RoboDK station: finished_products_shelf.rdk

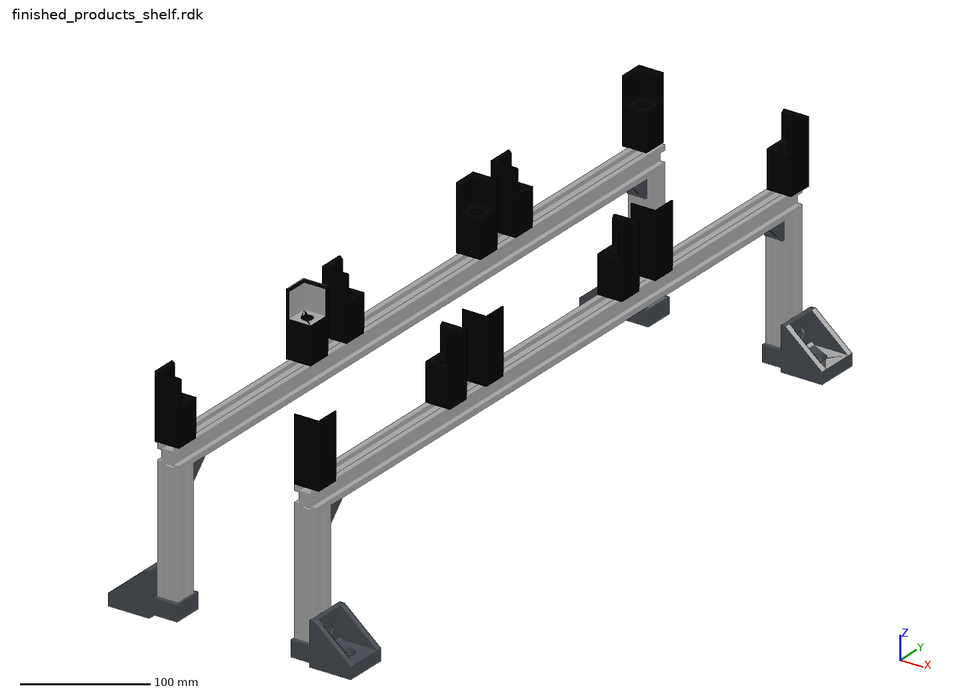
[picture v0: the station drawn from its stored meshes, robots at their saved joint values, targets as dots, program paths as lines]
Station final_deposit (saved by RoboDK 5.9.0). Poses are relative to the parent item; angles as X-Y-Z fixed-axis rotations.
  - object final_deposit at (0, 0, 0) mm, size 226.6 x 670.8 x 206.1 mm, geometry from final_deposit.stl
